{attribute 'qualified_only'}
{attribute 'strict'}
TYPE E_ExampleDeviceStates :
(
	enum_member := 0
);
END_TYPE

(* stored: Version 1.1.0.1, ProductVersion 3.1.4022.10
   DUT E_ExampleDeviceStates: Id {d3e11811-072d-49cd-b278-eb2789aaeb03} *)
